FUNCTION_BLOCK GO_TO_BLOW
VAR_INPUT
	xTransRelease:		BOOL;
END_VAR
VAR_OUTPUT
	xDone:			BOOL;
END_VAR
VAR
	lrTargetPos:		LREAL;
	xTransCondition:	BOOL;
	ftTimePulse:		F_TRIG;
	tpTimePulse:		TP;
END_VAR

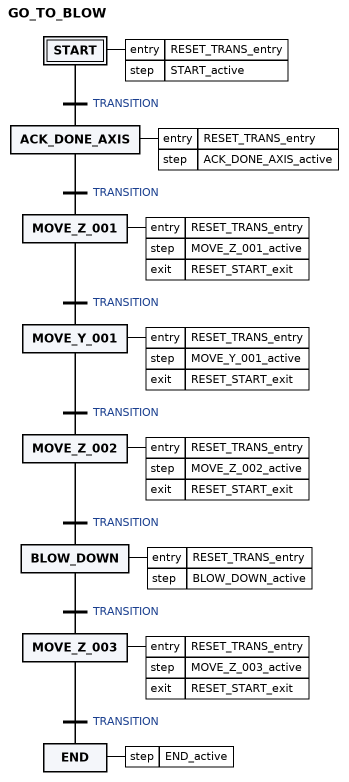
INITIAL_STEP START:
    RESET_TRANS_entry(P1);  // entry action
    START_active(N);  // step action
END_STEP
TRANSITION FROM START TO ACK_DONE_AXIS
    := TRANSITION;
END_TRANSITION
STEP ACK_DONE_AXIS:
    RESET_TRANS_entry(P1);  // entry action
    ACK_DONE_AXIS_active(N);  // step action
END_STEP
TRANSITION FROM ACK_DONE_AXIS TO MOVE_Z_001
    := TRANSITION;
END_TRANSITION
STEP MOVE_Z_001:
    RESET_TRANS_entry(P1);  // entry action
    MOVE_Z_001_active(N);  // step action
    RESET_START_exit(P0);  // exit action
END_STEP
TRANSITION FROM MOVE_Z_001 TO MOVE_Y_001
    := TRANSITION;
END_TRANSITION
STEP MOVE_Y_001:
    RESET_TRANS_entry(P1);  // entry action
    MOVE_Y_001_active(N);  // step action
    RESET_START_exit(P0);  // exit action
END_STEP
TRANSITION FROM MOVE_Y_001 TO MOVE_Z_002
    := TRANSITION;
END_TRANSITION
STEP MOVE_Z_002:
    RESET_TRANS_entry(P1);  // entry action
    MOVE_Z_002_active(N);  // step action
    RESET_START_exit(P0);  // exit action
END_STEP
TRANSITION FROM MOVE_Z_002 TO BLOW_DOWN
    := TRANSITION;
END_TRANSITION
STEP BLOW_DOWN:
    RESET_TRANS_entry(P1);  // entry action
    BLOW_DOWN_active(N);  // step action
END_STEP
TRANSITION FROM BLOW_DOWN TO MOVE_Z_003
    := TRANSITION;
END_TRANSITION
STEP MOVE_Z_003:
    RESET_TRANS_entry(P1);  // entry action
    MOVE_Z_003_active(N);  // step action
    RESET_START_exit(P0);  // exit action
END_STEP
TRANSITION FROM MOVE_Z_003 TO END
    := TRANSITION;
END_TRANSITION
STEP END:
    END_active(N);  // step action
END_STEP

ACTION ACK_DONE_AXIS_active:
IF G_sAxisDone.X OR G_sAxisDone.Y OR G_sAxisDone.Z OR G_sAxisDone.c THEN
	G_sAckAxisDone.X:=TRUE;
	G_sAckAxisDone.Y:=TRUE;
	G_sAckAxisDone.Z:=TRUE;
	G_sAckAxisDone.C:=TRUE;
ELSE
	G_sAckAxisDone.X:=FALSE;
	G_sAckAxisDone.Y:=FALSE;
	G_sAckAxisDone.Z:=FALSE;
	G_sAckAxisDone.C:=FALSE;
END_IF

xTransCondition:= NOT G_sAckAxisDone.X AND NOT G_sAckAxisDone.Y AND NOT G_sAckAxisDone.Z AND NOT G_sAckAxisDone.C;
END_ACTION

ACTION BLOW_DOWN_active:
tpTimePulse(IN:=NOT tpTimePulse.Q, PT:=T#500MS);
ftTimePulse(CLK:=tpTimePulse.Q);
xTransCondition:= ftTimePulse.Q;
END_ACTION

ACTION END_active:
xDone:=True;
END_ACTION

ACTION MOVE_Y_001_active:
G_sTargetPosition.Y:= G_asIndividualAxisPositions[CE_AXIS_Y].Positions[1].Target;
G_sStartToPos.Y:= TRUE;

xTransCondition:= G_sAxisDone.Y;
END_ACTION

ACTION MOVE_Z_001_active:
G_sTargetPosition.Z:= G_asIndividualAxisPositions[CE_AXIS_Z].Positions[1].Target;
G_sStartToPos.Z:= TRUE;

xTransCondition:= G_sAxisDone.Z;
END_ACTION

ACTION MOVE_Z_002_active:
G_sTargetPosition.Z:= G_asIndividualAxisPositions[CE_AXIS_Z].Positions[2].Target;
G_sStartToPos.Z:= TRUE;

xTransCondition:= G_sAxisDone.Z;
END_ACTION

ACTION MOVE_Z_003_active:
G_sTargetPosition.Z:= G_asIndividualAxisPositions[CE_AXIS_Z].Positions[1].Target;
G_sStartToPos.Z:= TRUE;

xTransCondition:= G_sAxisDone.Z;
END_ACTION

ACTION RESET_START_exit:
IF G_sAxisDone.X OR G_sAxisDone.Y OR G_sAxisDone.Z OR G_sAxisDone.c THEN
	G_sAckAxisDone.X:=TRUE;
	G_sAckAxisDone.Y:=TRUE;
	G_sAckAxisDone.Z:=TRUE;
	G_sAckAxisDone.C:=TRUE;
ELSE
	G_sAckAxisDone.X:=FALSE;
	G_sAckAxisDone.Y:=FALSE;
	G_sAckAxisDone.Z:=FALSE;
	G_sAckAxisDone.C:=FALSE;
	
	G_sStartToPos.X:=FALSE;
	G_sStartToPos.Y:=FALSE;
	G_sStartToPos.Z:=FALSE;
	G_sStartToPos.C:=FALSE;
END_IF
END_ACTION

ACTION RESET_TRANS_entry:
xTransCondition:= false;
END_ACTION

ACTION START_active:
xDone:=FALSE;

xTransCondition:= NOT xDone;
END_ACTION

TRANSITION TRANSITION:
xTransRelease AND xTransCondition
END_TRANSITION

END_FUNCTION_BLOCK

(* stored: Version 1.1.0.1, ProductVersion 3.1.4022.18
   POU GO_TO_BLOW: Id {c2d496e1-a9f8-4ceb-956a-04ffccdb8321}, SpecialFunc None
   Folder Active: Id {ae13b7f5-a8b1-422a-b577-3f4c89878efb}
   Folder Entry: Id {b6b5fe76-6e8b-46f6-b313-01af6e490efb}
   Folder Exit: Id {d1673ef2-f1fb-41a4-bede-b894d78d7af6}
   Folder Trans: Id {1542394e-9957-4fa6-b462-eaf2f74c5fa3}
   Action ACK_DONE_AXIS_active: Id {5ce54518-a0d9-4ac3-a7f8-cb42e49d4d0d}
   Action BLOW_DOWN_active: Id {43968463-dc20-4009-a839-b5a956100b1c}
   Action END_active: Id {32db9b5c-cfac-4f1a-a0b3-de4d2a15a7b7}
   Action MOVE_Y_001_active: Id {8e0f5470-23d5-48f3-96d4-e00ddf96c61f}
   Action MOVE_Z_001_active: Id {48e385ba-c2bb-4631-9895-2fb8d286f7dc}
   Action MOVE_Z_002_active: Id {37b188ef-6df9-485e-b3b6-e4d0a14caa84}
   Action MOVE_Z_003_active: Id {4b49ec4f-b012-4d28-85d2-259ad67bdb57}
   Action RESET_START_exit: Id {f6c53ba4-069e-4727-a727-99428df653d8}
   Action RESET_TRANS_entry: Id {1a2cb8ea-239e-4a3a-8cc8-08db21acec3b}
   Action START_active: Id {48f7c749-3596-45d8-b9f8-b44b92242723}
   Transition TRANSITION: Id {24f7ffcc-0565-4ad1-87bc-2f06f0ce77bd} *)
